(* Schneider Machine Expert - Basic project A11 Contador Descarga de Ar, file version 2.7.0.0 *)
(* ProjectInformations: Name=Novo projeto *)

HARDWARE
  Cpu 0: TM221M16R/G
  EthernetConfiguration: NetworkName=M221, IpAllocationMode=FixedAddress, IpAddress=0.0.0.0, SubnetMask=0.0.0.0
  SerialLineConfiguration: Baud=Baud19200, Parity=ParityEven, DataBits=DataBits8, StopBits=StopBits1, PhysicalMedium=PhysicalMediumRs485, TransmissionMode=TransmissionModeModbusRtu, SlaveId=1, Addressing=SlaveAddressing
  MastTask: UsePeriodScanMode=false, PeriodScan=100
  FastTask: Period=255
  CpuBehavior: StartingMode=StartAsPreviousState, AutoSaveRamOnEeprom=true, WatchdogPeriod=250

SYMBOLS  (address, symbol, comment, settings)
  %M0         "Habilita Pulso Ar"
  %M1         "Descarga de Ar"
  %TM0        [Preset=1, Base=OneSecond]
  %C0         [Preset=10]
  %C1         [Preset=1]
  %I0.0       "Chave Desliga"
  %I0.1       "Chave liga Ar"
  %Q0.0       "Valvula Puls Ar"

POU Novo POU
  (* SectionNumber=1 *)

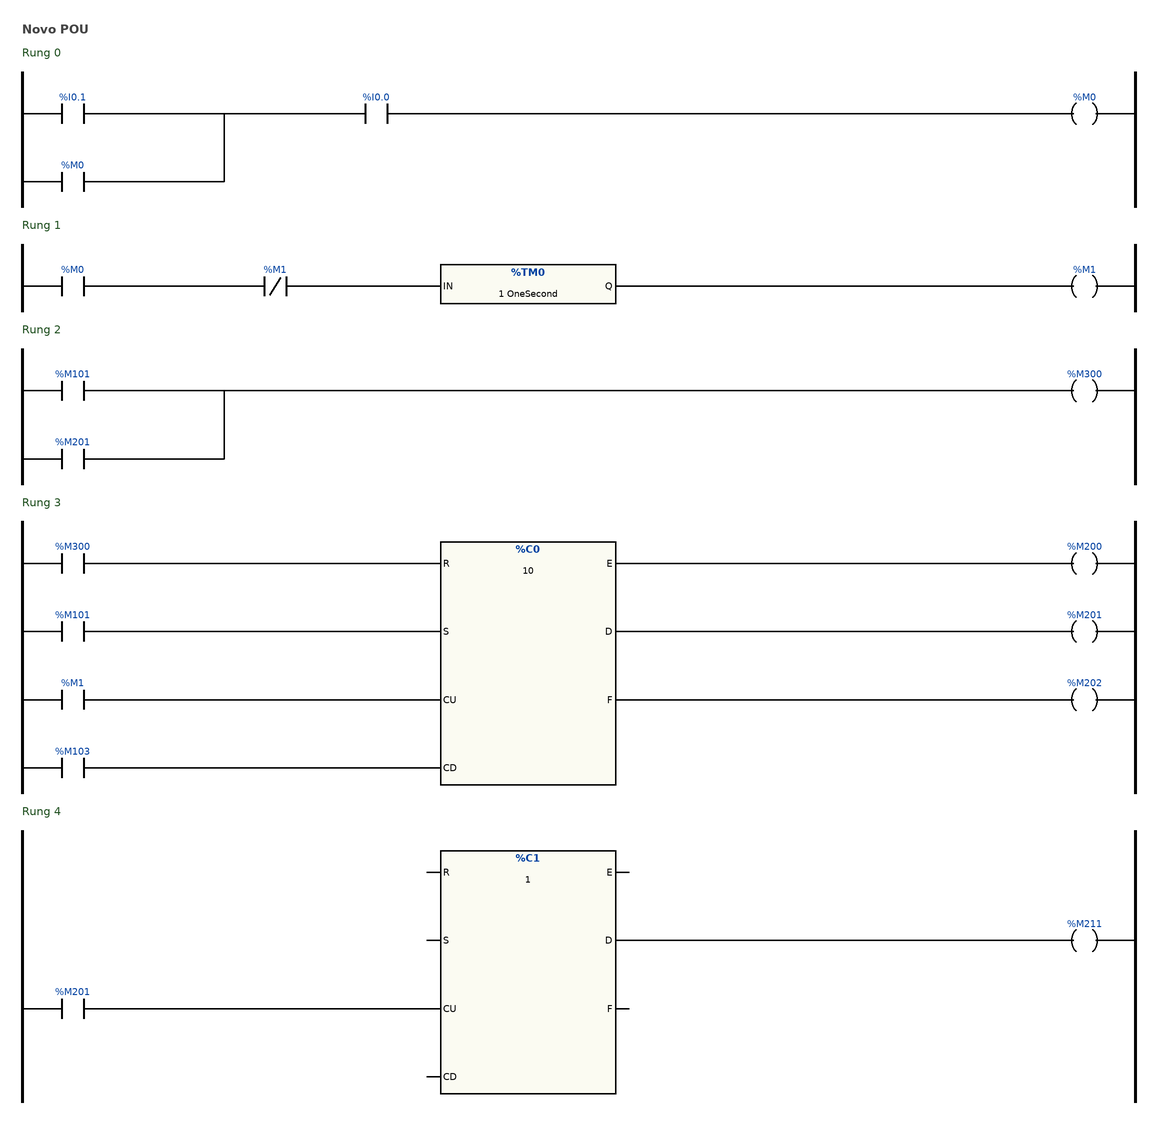

// Rung 0
  LD %I0.1
  OR %M0
  AND %I0.0
  ST %M0
  // as ST:
  //   %M0 := (%I0.1 OR %M0) AND %I0.0;

// Rung 1
  BLK %TM0
  LD %M0
  ANDN %M1
  IN
  OUT_BLK
  LD Q
  ST %M1
  END_BLK
  // as ST:
  //   %TM0(IN := %M0 AND NOT %M1);
  //   %M1 := %TM0.Q;

// Rung 2
  LD %M101
  OR %M201
  ST %M300
  // as ST:
  //   %M300 := %M101 OR %M201;

// Rung 3
  BLK %C0
  LD %M300
  R
  LD %M101
  S
  LD %M1
  CU
  LD %M103
  CD
  OUT_BLK
  LD E
  ST %M200
  LD D
  ST %M201
  LD F
  ST %M202
  END_BLK
  // as ST:
  //   %C0(R := %M300, S := %M101, CU := %M1, CD := %M103);
  //   %M200 := %C0.E;
  //   %M201 := %C0.D;
  //   %M202 := %C0.F;

// Rung 4
  BLK %C1
  LD %M201
  CU
  OUT_BLK
  LD D
  ST %M211
  END_BLK
  // as ST:
  //   %C1(CU := %M201);
  //   %M211 := %C1.D;
